// TIA Portal project "SuperSygnalizacjaDomiLechLuka" (V16)

(* hardware
DEVICE "S7-1200 station_2"  S7-1200 Station
   slot 0: "Rack_0"  S7-1200 Rack  Rack  V1.0
   slot 1: "PLC_2"  CPU 1215C AC/DC/Rly  6ES7 215-1BG40-0XB0  V4.4
DEVICE "S7-1200 station_1"  S7-1200 Station
   slot 0: "Rack_0"  S7-1200 Rack  Rack  V1.0
   slot 1: "PLC_1"  CPU 1215C AC/DC/Rly  6ES7 215-1BG40-0XB0  V4.4
*)

// ===== PLC "PLC_1"  CPU 1215C AC/DC/Rly =====

VAR_GLOBAL   // PLC tag table "Default tag table"
   "Clock_Byte" AT %MB0 : Byte;
   "Clock_10Hz" AT %M0.0 : Bool;
   "Clock_5Hz" AT %M0.1 : Bool;
   "Clock_2.5Hz" AT %M0.2 : Bool;
   "Clock_2Hz" AT %M0.3 : Bool;
   "Clock_1.25Hz" AT %M0.4 : Bool;
   "Clock_1Hz" AT %M0.5 : Bool;
   "Clock_0.625Hz" AT %M0.6 : Bool;
   "Clock_0.5Hz" AT %M0.7 : Bool;
   "P3_P4_green" AT %Q0.0 : Bool;
   "P3_P4_red" AT %Q0.1 : Bool;
   "W1_W3_W4_red" AT %Q0.2 : Bool;
   "W1_W3_W4_yellow" AT %Q0.3 : Bool;
   "W1_W3_W4_green" AT %Q0.4 : Bool;
   "W2_W6_red" AT %Q0.5 : Bool;
   "W2_W6_yellow" AT %Q0.6 : Bool;
   "W2_W6_green" AT %Q0.7 : Bool;
   "P2_red" AT %Q1.0 : Bool;
   "Start" AT %M3.0 : Bool;
   "Timer_CV" AT %MD10 : DWord;
END_VAR

DATA_BLOCK "sent"   // DB1
{ S7_Optimized_Access := 'FALSE' }
VERSION : 0.1
   VAR
      data : Bool;
   END_VAR
BEGIN
END_DATA_BLOCK

// folder: System blocks/Program resources

DATA_BLOCK "PLC_1_Send_DB"   // DB5
{ S7_Optimized_Access := 'TRUE' }
AUTHOR : SIMATIC
FAMILY : MC7Plus
NAME : TC_IP_v4
VERSION : 1.0
// stored: InstanceOfName TCON_IP_v4
"TCON_IP_v4"
BEGIN
   ID := 1;
   InterfaceId := 64;
   RemotePort := 2000;
   ActiveEstablished := true;
   RemoteAddress.ADDR[1] := 192;
   RemoteAddress.ADDR[2] := 168;
   RemoteAddress.ADDR[3] := 22;
   RemoteAddress.ADDR[4] := 138;
END_DATA_BLOCK

DATA_BLOCK "IEC_Timer_0_DB_1"   // DB6
{ S7_Optimized_Access := 'TRUE' }
AUTHOR : Simatic
FAMILY : IEC
NAME : IEC_TMR
VERSION : 1.0
// stored: InstanceOfName IEC_TIMER
"IEC_TIMER"
BEGIN
END_DATA_BLOCK

// folder: (top level)

ORGANIZATION_BLOCK "Main"   // OB1, LAD, ProgramCycle
TITLE = "Main Program Sweep (Cycle)"
{ S7_Optimized_Access := 'TRUE' }
VERSION : 0.1
   VAR_INPUT
      Initial_Call : Bool;   // Initial call of this OB
      Remanence : Bool;   // =True, if remanent data are available
   END_VAR
BEGIN

REGION Network 1
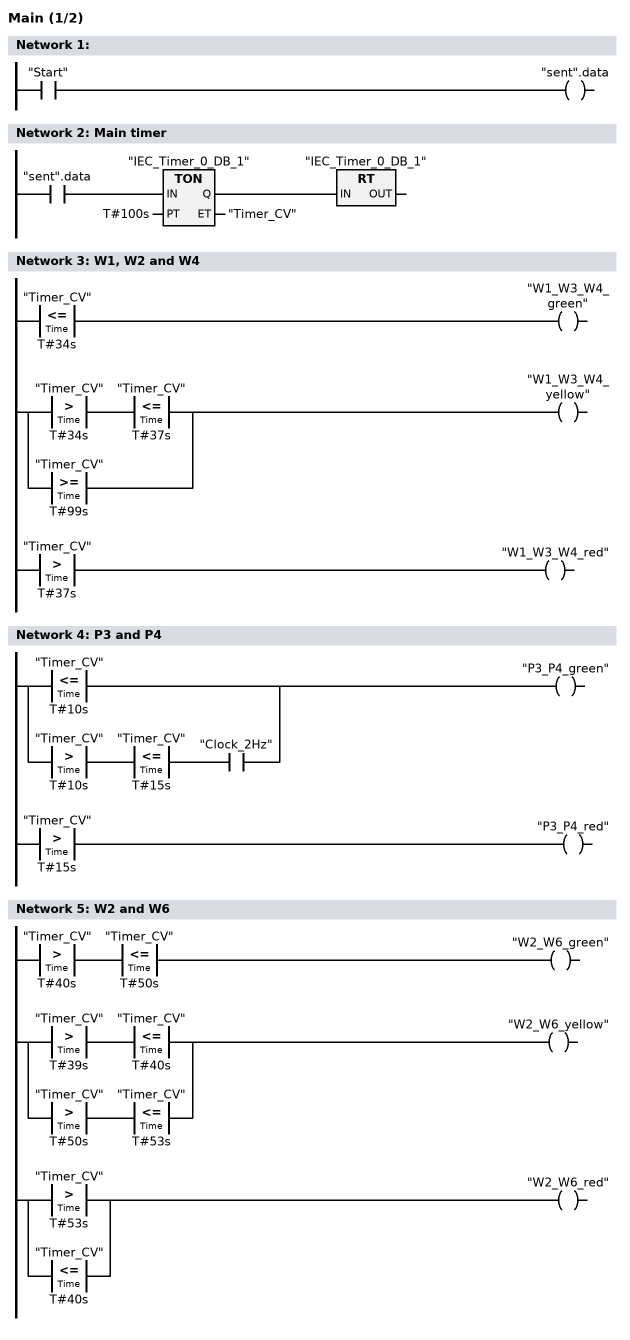
   RUNG wire#powerrail
      Contact( "Start" )
      Coil( "sent".data )
   END_RUNG
   // the same network as SCL:
   "sent".data := "Start";
END_REGION

REGION Network 2: Main timer
   "IEC_Timer_0_DB_1".TON(IN := "sent".data, PT := T#100s, ET => "Timer_CV");
   IF "IEC_Timer_0_DB_1".Q THEN RESET_TIMER("IEC_Timer_0_DB_1"); END_IF;
END_REGION

REGION Network 3: W1, W2 and W4
   RUNG wire#powerrail
      { S7_Templates := "SrcType := Time" } LE_Contact(in1 := "Timer_CV", in2 := T#34s)
      Coil( "W1_W3_W4_green" )
   END_RUNG
   RUNG wire#powerrail
      { S7_Templates := "SrcType := Time" } GT_Contact(in1 := "Timer_CV", in2 := T#34s)
      { S7_Templates := "SrcType := Time" } LE_Contact(in1 := "Timer_CV", in2 := T#37s)
      wire#w1
      Coil( "W1_W3_W4_yellow" )
   END_RUNG
   RUNG wire#powerrail
      { S7_Templates := "SrcType := Time" } GE_Contact(in1 := "Timer_CV", in2 := T#99s)
   END_RUNG wire#w1
   RUNG wire#powerrail
      { S7_Templates := "SrcType := Time" } GT_Contact(in1 := "Timer_CV", in2 := T#37s)
      Coil( "W1_W3_W4_red" )
   END_RUNG
   // the same network as SCL:
   "W1_W3_W4_green" := "Timer_CV" <= T#34s;
   "W1_W3_W4_yellow" := (("Timer_CV" > T#34s) AND ("Timer_CV" <= T#37s)) OR ("Timer_CV" >= T#99s);
   "W1_W3_W4_red" := "Timer_CV" > T#37s;
END_REGION

REGION Network 4: P3 and P4
   RUNG wire#powerrail
      { S7_Templates := "SrcType := Time" } LE_Contact(in1 := "Timer_CV", in2 := T#10s)
      wire#w1
      Coil( "P3_P4_green" )
   END_RUNG
   RUNG wire#powerrail
      { S7_Templates := "SrcType := Time" } GT_Contact(in1 := "Timer_CV", in2 := T#10s)
      { S7_Templates := "SrcType := Time" } LE_Contact(in1 := "Timer_CV", in2 := T#15s)
      Contact( "Clock_2Hz" )
   END_RUNG wire#w1
   RUNG wire#powerrail
      { S7_Templates := "SrcType := Time" } GT_Contact(in1 := "Timer_CV", in2 := T#15s)
      Coil( "P3_P4_red" )
   END_RUNG
   // the same network as SCL:
   "P3_P4_green" := ("Timer_CV" <= T#10s) OR (("Timer_CV" > T#10s) AND ("Timer_CV" <= T#15s) AND "Clock_2Hz");
   "P3_P4_red" := "Timer_CV" > T#15s;
END_REGION

REGION Network 5: W2 and W6
   RUNG wire#powerrail
      { S7_Templates := "SrcType := Time" } GT_Contact(in1 := "Timer_CV", in2 := T#40s)
      { S7_Templates := "SrcType := Time" } LE_Contact(in1 := "Timer_CV", in2 := T#50s)
      Coil( "W2_W6_green" )
   END_RUNG
   RUNG wire#powerrail
      { S7_Templates := "SrcType := Time" } GT_Contact(in1 := "Timer_CV", in2 := T#39s)
      { S7_Templates := "SrcType := Time" } LE_Contact(in1 := "Timer_CV", in2 := T#40s)
      wire#w1
      Coil( "W2_W6_yellow" )
   END_RUNG
   RUNG wire#powerrail
      { S7_Templates := "SrcType := Time" } GT_Contact(in1 := "Timer_CV", in2 := T#50s)
      { S7_Templates := "SrcType := Time" } LE_Contact(in1 := "Timer_CV", in2 := T#53s)
   END_RUNG wire#w1
   RUNG wire#powerrail
      { S7_Templates := "SrcType := Time" } GT_Contact(in1 := "Timer_CV", in2 := T#53s)
      wire#w2
      Coil( "W2_W6_red" )
   END_RUNG
   RUNG wire#powerrail
      { S7_Templates := "SrcType := Time" } LE_Contact(in1 := "Timer_CV", in2 := T#40s)
   END_RUNG wire#w2
   // the same network as SCL:
   "W2_W6_green" := ("Timer_CV" > T#40s) AND ("Timer_CV" <= T#50s);
   "W2_W6_yellow" := (("Timer_CV" > T#39s) AND ("Timer_CV" <= T#40s)) OR (("Timer_CV" > T#50s) AND ("Timer_CV" <= T#53s));
   "W2_W6_red" := ("Timer_CV" > T#53s) OR ("Timer_CV" <= T#40s);
END_REGION

REGION Network 6: P2
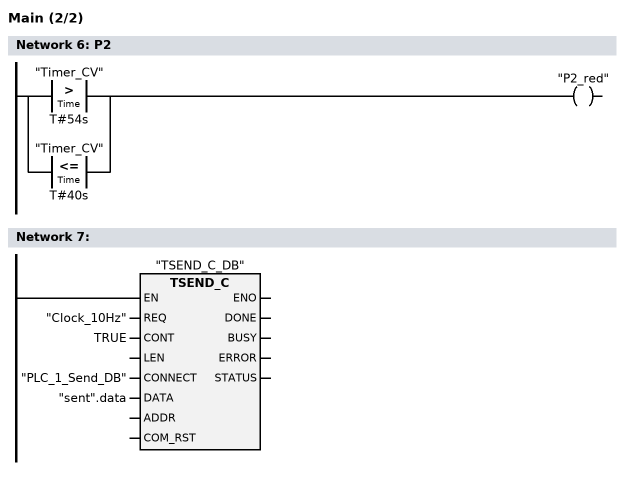
   RUNG wire#powerrail
      { S7_Templates := "SrcType := Time" } GT_Contact(in1 := "Timer_CV", in2 := T#54s)
      wire#w1
      Coil( "P2_red" )
   END_RUNG
   RUNG wire#powerrail
      { S7_Templates := "SrcType := Time" } LE_Contact(in1 := "Timer_CV", in2 := T#40s)
   END_RUNG wire#w1
   // the same network as SCL:
   "P2_red" := ("Timer_CV" > T#54s) OR ("Timer_CV" <= T#40s);
END_REGION

REGION Network 7
   "TSEND_C_DB"(REQ := "Clock_10Hz", CONT := TRUE, CONNECT := "PLC_1_Send_DB", DATA := "sent".data);   // TSEND_C
END_REGION
END_ORGANIZATION_BLOCK

// ===== PLC "PLC_2"  CPU 1215C AC/DC/Rly =====

VAR_GLOBAL   // PLC tag table "Default tag table"
   "Clock_Byte" AT %MB0 : Byte;
   "Clock_10Hz" AT %M0.0 : Bool;
   "Clock_5Hz" AT %M0.1 : Bool;
   "Clock_2.5Hz" AT %M0.2 : Bool;
   "Clock_2Hz" AT %M0.3 : Bool;
   "Clock_1.25Hz" AT %M0.4 : Bool;
   "Clock_1Hz" AT %M0.5 : Bool;
   "Clock_0.625Hz" AT %M0.6 : Bool;
   "Clock_0.5Hz" AT %M0.7 : Bool;
   "P2_green" AT %Q0.0 : Bool;
   "W7_red" AT %Q0.1 : Bool;
   "W7_yellow" AT %Q0.2 : Bool;
   "W7_green" AT %Q0.3 : Bool;
   "W5_red" AT %Q0.4 : Bool;
   "W5_yellow" AT %Q0.5 : Bool;
   "W5_green" AT %Q0.6 : Bool;
   "P1_red" AT %Q0.7 : Bool;
   "P1_green" AT %Q1.0 : Bool;
   "Timer_CV" AT %MD1 : DWord;
END_VAR

DATA_BLOCK "recv"   // DB2
{ S7_Optimized_Access := 'FALSE' }
VERSION : 0.1
   VAR
      data : Bool;
   END_VAR
BEGIN
END_DATA_BLOCK

// folder: System blocks/Program resources

DATA_BLOCK "IEC_Timer_0_DB"   // DB1
{ S7_Optimized_Access := 'TRUE' }
AUTHOR : Simatic
FAMILY : IEC
NAME : IEC_TMR
VERSION : 1.0
// stored: InstanceOfName IEC_TIMER
"IEC_TIMER"
BEGIN
END_DATA_BLOCK

DATA_BLOCK "PLC_2_Receive_DB"   // DB4
{ S7_Optimized_Access := 'TRUE' }
AUTHOR : SIMATIC
FAMILY : MC7Plus
NAME : TC_IP_v4
VERSION : 1.0
// stored: InstanceOfName TCON_IP_v4
"TCON_IP_v4"
BEGIN
   ID := 1;
   InterfaceId := 64;
   LocalPort := 2000;
   RemoteAddress.ADDR[1] := 192;
   RemoteAddress.ADDR[2] := 168;
   RemoteAddress.ADDR[3] := 22;
   RemoteAddress.ADDR[4] := 139;
END_DATA_BLOCK

// folder: (top level)

ORGANIZATION_BLOCK "Main"   // OB1, LAD, ProgramCycle
TITLE = "Main Program Sweep (Cycle)"
{ S7_Optimized_Access := 'TRUE' }
VERSION : 0.1
   VAR_INPUT
      Initial_Call : Bool;   // Initial call of this OB
      Remanence : Bool;   // =True, if remanent data are available
   END_VAR
BEGIN

REGION Network 1
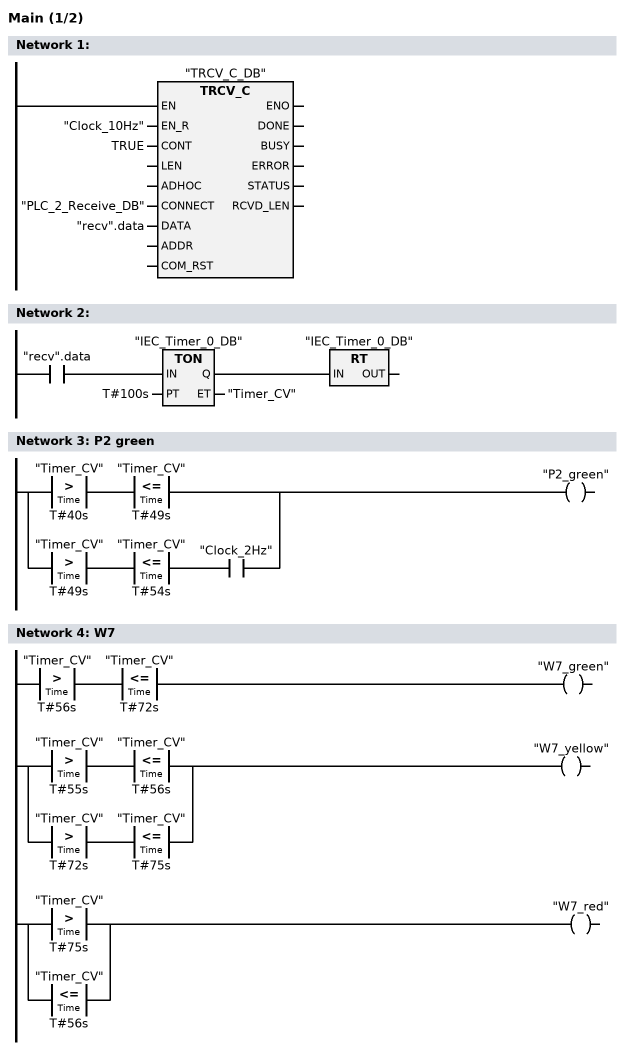
   "TRCV_C_DB"(EN_R := "Clock_10Hz", CONT := TRUE, CONNECT := "PLC_2_Receive_DB", DATA := "recv".data);   // TRCV_C
END_REGION

REGION Network 2
   "IEC_Timer_0_DB".TON(IN := "recv".data, PT := T#100s, ET => "Timer_CV");
   IF "IEC_Timer_0_DB".Q THEN RESET_TIMER("IEC_Timer_0_DB"); END_IF;
END_REGION

REGION Network 3: P2 green
   RUNG wire#powerrail
      { S7_Templates := "SrcType := Time" } GT_Contact(in1 := "Timer_CV", in2 := T#40s)
      { S7_Templates := "SrcType := Time" } LE_Contact(in1 := "Timer_CV", in2 := T#49s)
      wire#w1
      Coil( "P2_green" )
   END_RUNG
   RUNG wire#powerrail
      { S7_Templates := "SrcType := Time" } GT_Contact(in1 := "Timer_CV", in2 := T#49s)
      { S7_Templates := "SrcType := Time" } LE_Contact(in1 := "Timer_CV", in2 := T#54s)
      Contact( "Clock_2Hz" )
   END_RUNG wire#w1
   // the same network as SCL:
   "P2_green" := (("Timer_CV" > T#40s) AND ("Timer_CV" <= T#49s)) OR (("Timer_CV" > T#49s) AND ("Timer_CV" <= T#54s) AND "Clock_2Hz");
END_REGION

REGION Network 4: W7
   RUNG wire#powerrail
      { S7_Templates := "SrcType := Time" } GT_Contact(in1 := "Timer_CV", in2 := T#56s)
      { S7_Templates := "SrcType := Time" } LE_Contact(in1 := "Timer_CV", in2 := T#72s)
      Coil( "W7_green" )
   END_RUNG
   RUNG wire#powerrail
      { S7_Templates := "SrcType := Time" } GT_Contact(in1 := "Timer_CV", in2 := T#55s)
      { S7_Templates := "SrcType := Time" } LE_Contact(in1 := "Timer_CV", in2 := T#56s)
      wire#w1
      Coil( "W7_yellow" )
   END_RUNG
   RUNG wire#powerrail
      { S7_Templates := "SrcType := Time" } GT_Contact(in1 := "Timer_CV", in2 := T#72s)
      { S7_Templates := "SrcType := Time" } LE_Contact(in1 := "Timer_CV", in2 := T#75s)
   END_RUNG wire#w1
   RUNG wire#powerrail
      { S7_Templates := "SrcType := Time" } GT_Contact(in1 := "Timer_CV", in2 := T#75s)
      wire#w2
      Coil( "W7_red" )
   END_RUNG
   RUNG wire#powerrail
      { S7_Templates := "SrcType := Time" } LE_Contact(in1 := "Timer_CV", in2 := T#56s)
   END_RUNG wire#w2
   // the same network as SCL:
   "W7_green" := ("Timer_CV" > T#56s) AND ("Timer_CV" <= T#72s);
   "W7_yellow" := (("Timer_CV" > T#55s) AND ("Timer_CV" <= T#56s)) OR (("Timer_CV" > T#72s) AND ("Timer_CV" <= T#75s));
   "W7_red" := ("Timer_CV" > T#75s) OR ("Timer_CV" <= T#56s);
END_REGION

REGION Network 5: W5
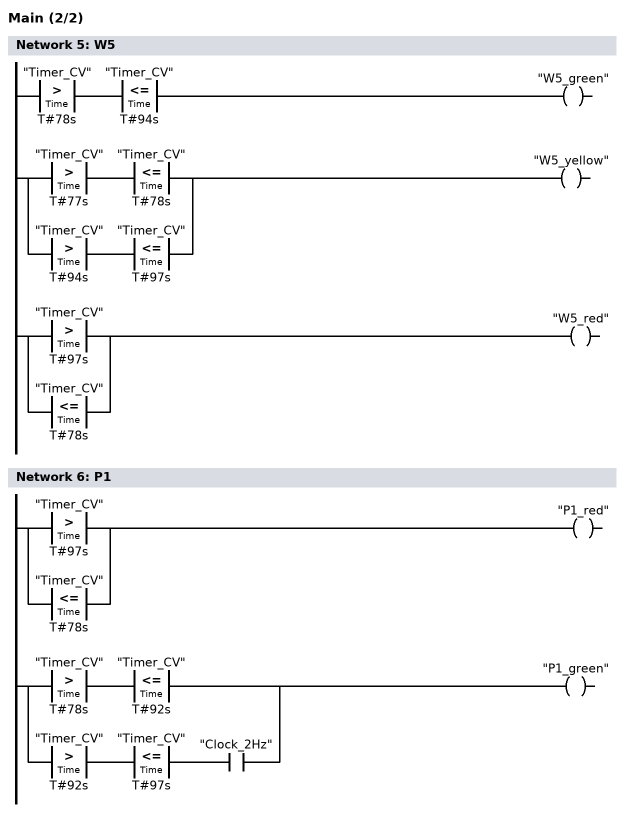
   RUNG wire#powerrail
      { S7_Templates := "SrcType := Time" } GT_Contact(in1 := "Timer_CV", in2 := T#78s)
      { S7_Templates := "SrcType := Time" } LE_Contact(in1 := "Timer_CV", in2 := T#94s)
      Coil( "W5_green" )
   END_RUNG
   RUNG wire#powerrail
      { S7_Templates := "SrcType := Time" } GT_Contact(in1 := "Timer_CV", in2 := T#77s)
      { S7_Templates := "SrcType := Time" } LE_Contact(in1 := "Timer_CV", in2 := T#78s)
      wire#w1
      Coil( "W5_yellow" )
   END_RUNG
   RUNG wire#powerrail
      { S7_Templates := "SrcType := Time" } GT_Contact(in1 := "Timer_CV", in2 := T#94s)
      { S7_Templates := "SrcType := Time" } LE_Contact(in1 := "Timer_CV", in2 := T#97s)
   END_RUNG wire#w1
   RUNG wire#powerrail
      { S7_Templates := "SrcType := Time" } GT_Contact(in1 := "Timer_CV", in2 := T#97s)
      wire#w2
      Coil( "W5_red" )
   END_RUNG
   RUNG wire#powerrail
      { S7_Templates := "SrcType := Time" } LE_Contact(in1 := "Timer_CV", in2 := T#78s)
   END_RUNG wire#w2
   // the same network as SCL:
   "W5_green" := ("Timer_CV" > T#78s) AND ("Timer_CV" <= T#94s);
   "W5_yellow" := (("Timer_CV" > T#77s) AND ("Timer_CV" <= T#78s)) OR (("Timer_CV" > T#94s) AND ("Timer_CV" <= T#97s));
   "W5_red" := ("Timer_CV" > T#97s) OR ("Timer_CV" <= T#78s);
END_REGION

REGION Network 6: P1
   RUNG wire#powerrail
      { S7_Templates := "SrcType := Time" } GT_Contact(in1 := "Timer_CV", in2 := T#97s)
      wire#w1
      Coil( "P1_red" )
   END_RUNG
   RUNG wire#powerrail
      { S7_Templates := "SrcType := Time" } LE_Contact(in1 := "Timer_CV", in2 := T#78s)
   END_RUNG wire#w1
   RUNG wire#powerrail
      { S7_Templates := "SrcType := Time" } GT_Contact(in1 := "Timer_CV", in2 := T#78s)
      { S7_Templates := "SrcType := Time" } LE_Contact(in1 := "Timer_CV", in2 := T#92s)
      wire#w2
      Coil( "P1_green" )
   END_RUNG
   RUNG wire#powerrail
      { S7_Templates := "SrcType := Time" } GT_Contact(in1 := "Timer_CV", in2 := T#92s)
      { S7_Templates := "SrcType := Time" } LE_Contact(in1 := "Timer_CV", in2 := T#97s)
      Contact( "Clock_2Hz" )
   END_RUNG wire#w2
   // the same network as SCL:
   "P1_red" := ("Timer_CV" > T#97s) OR ("Timer_CV" <= T#78s);
   "P1_green" := (("Timer_CV" > T#78s) AND ("Timer_CV" <= T#92s)) OR (("Timer_CV" > T#92s) AND ("Timer_CV" <= T#97s) AND "Clock_2Hz");
END_REGION
END_ORGANIZATION_BLOCK